RoboDK station: My_Bachelor_Project_Sim.rdk

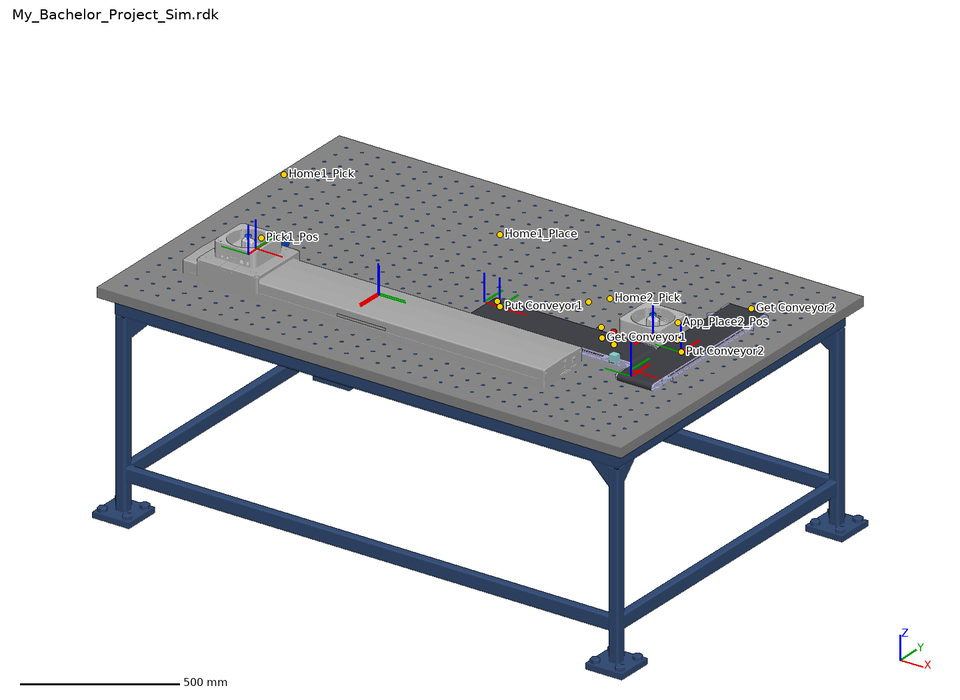
[picture v0: the station drawn from its stored meshes, robots at their saved joint values, targets as dots, program paths as lines]
Station My_Bachelor_Project_Sim (saved by RoboDK 5.9.2). Poses are relative to the parent item; angles as X-Y-Z fixed-axis rotations.
  - object Table  at (0, 0, 0) mm, size 2020 x 1340 x 800 mm, geometry from Table-2000x1200x800mm.sld
    - frame Conveyor1_frame at (730, -120, 40) mm
      - object Conveyor1 at (520, -80, -20) mm, rotated rx 0 ry 0 rz 90 deg, size 179.1 x 627.2 x 32.2 mm
      - frame Conveyor_1 Base at (0, 0, 0) mm
        - robot Conveyor_1: 1 axes
            modified DH rows (alpha deg, a mm, theta deg, d mm): 0, 0, 0, 0 linear
            base shift (0, 0, 0) mm, rotated rx 0 ry 90 rz 0 deg
            joint limits [0] to [600]; home [0]; saved at [0]
      - target Put Conveyor1 (Cartesian target) at (59.25, 0, -0.79) mm; joints [134.006, 22.86, -66.558, 43.699, -45.994, 0]
      - target Get Conveyor1 (Cartesian target) at (450, 0, 0) mm; joints [0, 0, 0, 0, 0, 43.699]
      - object Motion_Sensor at (450, 62, 20) mm, size 18 x 18 x 24 mm
      - object Colour_Sensor at (550, -108, -10) mm, size 25.9 x 25.9 x 25.9 mm, geometry from Cube-50mm (1).sld
      - frame Put_Conveyor1_Frame at (60, 0, 0) mm
        - target Home1_Place (Cartesian target) at (0, 0, 250) mm, rotated rx 180 ry 0 rz -90 deg; joints [0, 0, 0, 0] of Dobot Magician1
        - target Place1_Pos (Cartesian target) at (4.5, -22, 29.12) mm, rotated rx 180 ry 0 rz -90 deg; joints [-2.421, 65.885, 80.616, -2.421] of Dobot Magician1
    - frame Conveyor2_Frame at (1360, -220, 20) mm
      - frame Put_Conveyor2_Frame at (80, 160, 20) mm, rotated rx 0 ry 0 rz 90 deg
        - target Put Conveyor2 (Cartesian target) at (0, 0, 0) mm; joints [134.006, 22.86, -66.558, 43.699, -45.994, 0]
        - target Get Conveyor2 (Cartesian target) at (380, 0, 0) mm; joints [0, 0, 0, 0, 0, 43.699]
      - object Conveyor2 at (0, 0, 0) mm, size 179.1 x 627.2 x 32.2 mm
      - frame Conveyor_2 Base at (50, -70, 20) mm, rotated rx 0 ry 0 rz 90 deg
        - robot Conveyor_2: 1 axes
            modified DH rows (alpha deg, a mm, theta deg, d mm): 0, 0, 0, 0 linear
            base shift (0, 0, 0) mm, rotated rx 0 ry 90 rz 0 deg
            joint limits [0] to [600]; home [0]; saved at [380]
  - frame Rail_Reference at (480, -340, 90) mm, rotated rx 0 ry 0 rz -90 deg
    - frame Linear Rail Base at (10, 10, 0) mm
      - robot Linear Rail  (model Brooks PreciseFlex Linear Rail 1000): 1 axes
          modified DH rows (alpha deg, a mm, theta deg, d mm): 0, 0, 0, 0 linear
          base shift (0, 0, 0) mm, rotated rx 0 ry 90 rz 90 deg
          joint limits [-500] to [500]; home [0]; saved at [-500]
        - frame Dobot Magician1 Base at (0, 0, 1) mm, rotated rx 0 ry 0 rz -180 deg
          - robot Dobot Magician1 (model Dobot Magician): 4 axes, payload 0.5 kg, reach 320 mm, repeatability 0.2 mm, weight 4 kg
              joint limits [-90, -0.001, -10, -90] to [90, 85, 95, 90]; home [0, 0, 0, 0]; saved at [-26.105, 17.869, 35.082, 63.895]
            - tool Vacuum Gripper1, TCP at (0, 0, 65) mm, size 37.5 x 41.5 x 68.1 mm
      - target Rail_Home (Cartesian target) at (0, 0, 0) mm; joints [0] of Linear Rail 
      - target Rail_Pick_Pos (Cartesian target) at (0, -500, 0) mm; joints [-500] of Linear Rail 
      - target Rail_Place_Pos (Cartesian target) at (0, 295.7, 0) mm; joints [295.7] of Linear Rail 
  - frame Box_Frame at (-120, -150, 0) mm
    - object Red_Cube at (50, 0, 0) mm, size 25 x 25 x 25 mm, geometry from Cube-50mm (1).sld
    - object Green_Cube at (0, 50, 0) mm, size 25 x 25 x 25 mm, geometry from Cube-50mm (1).sld
    - object Blue_Cube at (50, 50, 0) mm, size 25 x 25 x 25 mm, geometry from Cube-50mm (1).sld
    - target Home1_Pick (Cartesian target) at (100, 10, 280) mm, rotated rx 180 ry 0 rz -90 deg; joints [2.726, 1.232, 5.453, 2.726] of Dobot Magician1
    - target Pick1_Pos (Cartesian target) at (13.34, 10.05, 37.21) mm, rotated rx 180 ry 0 rz -90 deg; joints [24.71, 81.254, 75.504, 24.71] of Dobot Magician1
    - object yellow_Cube at (0, 0, 0) mm, size 25 x 25 x 25 mm, geometry from Cube-50mm (1).sld
  - frame Dobot Magician2 Base at (1240, 70, 0) mm, rotated rx 0 ry 0 rz -90 deg
    - robot Dobot Magician2 (model Dobot Magician): 4 axes, payload 0.5 kg, reach 320 mm, repeatability 0.2 mm, weight 4 kg
        joint limits [-90, -0.001, -10, -90] to [90, 85, 95, 90]; home [0, 0, 0, 0]; saved at [0, 10.83, -4.63, 0]
      - tool Vacuum Gripper2, TCP at (0, 0, 65) mm, size 37.5 x 41.5 x 68.1 mm
    - target Home2_Pick (Cartesian target) at (232.89, 0, 212.46) mm, rotated rx 180 ry 0 rz -180 deg; joints [0, 10.83, -4.63, 0] of Dobot Magician2
    - target App_Pick2_Pos (Cartesian target) at (245.79, -71.87, 184.7) mm, rotated rx 180 ry 0 rz 163.7 deg; joints [-16.3, 21, 3.64, 0] of Dobot Magician2
    - target Pick2_Pos (Cartesian target) at (196.48, -57.46, 81.24) mm, rotated rx 180 ry 0 rz 163.7 deg; joints [-16.3, 21.33, 49.94, 0] of Dobot Magician2
    - target Sensor_Place2_Pos (Cartesian target) at (287.45, 53.95, 89.18) mm, rotated rx 180 ry 0 rz -169.37 deg; joints [10.63, 48.57, 27.62, 0] of Dobot Magician2
    - target App_Place2_Pos (Cartesian target) at (124.89, 185.02, 137.37) mm, rotated rx 180 ry 0 rz -124.02 deg; joints [55.98, 12.47, 25.14, 0] of Dobot Magician2
    - target Place2_Pos (Cartesian target) at (124.99, 180.37, 74.44) mm, rotated rx 180 ry 0 rz -124.72 deg; joints [55.28, 28.22, 49.94, 0] of Dobot Magician2
  - Python program Dobot_1_Prog (listed below)
  - Python program Dobot_2_Prog (listed below)
  - Python program Conveyor_1_Prog (listed below)
  - Python program Conveyor_2_Prog (listed below)
  - Python program Main_Common_Prog (listed below)

--- Python program Dobot_1_Prog ---
# Link to RoboDK
#### Dobot1 Programme ####

from robolink import *
from robodk import *
from time import sleep
sim = robolink.Robolink()

#Items
base = sim.Item("Dobot Magician1 Base")
robot1 = sim.Item("Dobot Magician1")
tool1 = sim.Item("Vacuum Gripper1")


#Conveyors
conveyor1 = sim.Item("Conveyor Belt1")


if not robot1.Valid():
    raise Exception("Robot not found")
if not tool1.Valid():
    raise Exception("Tool not found")

#frames
baseFrame = sim.Item("Dobot Magician1 Base")
rail = sim.Item("Linear Rail", ITEM_TYPE_ROBOT)
pickFrame =sim.Item("Box_Frame")
putFrame  = sim.Item("Put_Conveyor1_Frame")

# Targets
home1_Pick = sim.Item("Home1_Pick")
home1_Place = sim.Item("Home1_Place")
#app_Pick_Pos = sim.Item("App_Pick_Pos")
#app_Place_Pos = sim.Item("App__Place_Pos")
pick_Pos = sim.Item("Pick_Pos")
place_Pos = sim.Item("Place_Pos")

#objects
box1 = sim.Item("Yellow_Cube")
box2= sim.Item("Red_Cube")
box3 = sim.Item("Green_Cube")
box4 = sim.Item("Blue_Cube")
conveyor_Frame = sim.Item("Conveyro_Box_Frame")

# Targets (RAIL)

rail_home  = sim.Item("Rail_Home")
rail_pick  = sim.Item("Rail_Pick_Pos")
rail_place = sim.Item("Rail_Place_Pos")

for item in [rail_home, rail_pick, rail_place, app_pos_Pick, app_Pos_Place, pick_Pos, place_Pos]:
    if not item.Valid():
        raise Exception(f"Missing item: {item.Name()}")

robot1.setSpeed(200,50)
robot1.setPoseTool(tool1)

robot1.setPoseFrame(baseFrame)
rail.MoveJ(rail_home)
rail.MoveJ(rail_pick)

#Pick
robot1.setPoseFrame(pickFrame)
box.setParentStatic(pickFrame)
robot1.MoveJ(app_pos_Pick)
robot1.MoveJ(pick_Pos)
tool1.AttachClosest()
robot1.MoveJ(app_pos_Pick)

#Move to Put
robot1.setPoseFrame(baseFrame)
rail.MoveJ(rail_place)

#Put
robot1.setPoseFrame(putFrame)
robot1.MoveJ(app_Pos_Place)
robot1.MoveJ(place_Pos)
tool1.DetachAll()
box.setParent(putFrame)
box.setParentStatic(conveyor1)
robot1.MoveJ(app_Pos_Place)

robot1.setPoseFrame(baseFrame)
rail.MoveJ(rail_home)

--- Python program Dobot_2_Prog ---
from robolink import *
from robodk import *
sim = robolink.Robolink()

#Items
base2 = sim.Item("Dobot Magician2 Base")
robot2 = sim.Item("Dobot Magician2")
tool2  = sim.Item("Vacuum Gripper2")
conveyor1 = sim.Item("Conveyor1")
conveyor2 = sim.Item("Conveyor")
box = sim.Item("Cube_Box")

# Frames
box_Frame_Pick = sim.Item("Conv1_Box_Frame")
box_Frame_Put = sim.Item("Conv2_Box_Frame")

# Targets
home2 = sim.Item("Home_Dobot2")
app_Pick_Conv1 = sim.Item("App_Pick_Pose_Conv1")
Pick_Conv1 = sim.Item("Pick_Pos_Conv1")
app_put_Conv2 = sim.Item("App_Put_Box_Conv2")
put_Conv2 = sim.Item("Put_Box_Conv2")


base = sim.Item("Dobot Magician2 Base")

# Gå to the conveyor and pick the cube

robot2.setSpeed(200,50)

# go to home for dobot2 base frame
robot2.setFrame(base2)
robot2.MoveJ(home2)

# go to pick position
robot2.setTool(tool2)
robot2.setFrame(base2)
robot2.MoveJ(app_Pick_Conv1)
robot2.MoveJ(Pick_Conv1)

# attach cube
box.setParent(box_Frame_Pick)
tool2.AttachClosest()

# go to put position
robot2.MoveJ(app_put_Conv2)
robot2.MoveJ(put_Conv2)
box.setParent(conveyor2)
tool2.DetachAll()

robot2.setFrame(base2)
robot2.MoveJ(home2)

--- Python program Conveyor_1_Prog ---
#### Conveyor1 programme ####

# To connect with the RoboDK
from robolink import *
from robodk import *
from time import sleep

sim = robolink.Robolink()

# Item
conveyor1 = sim.Item("Conveyor Belt1")
box = sim.Item("Cube")

# Frame
conveyor1_Frame = sim.Item("Conveyor Belt1 Base")
conveyorReference = sim.Item("ConveyorReference")
put_Conveyor1_Frame = sim.Item("Put_Conveyor1_Frame", ITEM_TYPE_FRAME)

# Targets
put_pos = sim.Item("Put Conveyor1")
get_pos = sim.Item("Get Conveyor1")

if not conveyor1.Valid() or not box.Valid():
    raise Exception("Items not found")

# Programme to set or atach the box ti the put_pos
# Attach cube to Put Conveyor1

all_items = sim.ItemList()
for item in all_items:
    print(item.Name())

def run_cycle():

    if not put_Conveyor1_Frame.Valid():
        raise Exception("Put_Conveyor1_Frame not found")

    box.setParentStatic(put_Conveyor1_Frame)
    box.setPose(transl(0,0,0,))

    box.setParentStatic(conveyor1)
    sleep(0.1)

     # Move conveyor slowly
    for i in range(0,1500,20):   # step size controls speed
        conveyor1.setJoints([i])
        sleep(0.05)
    print("Conveyor1 cycle complete")

 # Run 5 times again
print("Starting 5-run loop...")
for i in range(2):
    print(f"Iteration {i+1}")
    run_cycle()
    sleep(0.5)

--- Python program Conveyor_2_Prog ---
#### Conveyor2 programme ####

# To connect with the RoboDK
from robolink import *
from robodk import *
from time import sleep

sim = robolink.Robolink()

# Item
conveyor2 = sim.Item("Conveyor Belt2")
box_frame = sim.Item("Put_Conv2")
box = sim.Item("Cube_Box")

# Check validity
if not box.Valid():
    raise Exception("Check! cube not found")

#Targets
home_pos = sim.Item("Conv2_Home_Put")
yellow_pos = sim.Item("Get_Conv2_Yellow")
non_yellow_pos =sim.Item("Get_Conv2_Non_Yellow")

if not home_pos.Valid() or not yellow_pos.Valid() or not non_yellow_pos.Valid():
    raise Exception("Check target names")

# Reset conveyor
box.setParentStatic(conveyor2)
sleep(0.1)

#conveyor2.MoveJ(home_pos)
#sleep(0.3)
cube_colour = "yellow"
#cube_colour = "red"
#cube_colour = "green"
#cube_colour = "blue"


# Move depending on colour
if cube_colour == "yellow":
    conveyor2.MoveJ(yellow_pos)
else:
    conveyor2.MoveJ(non_yellow_pos)

sleep(0.5)

conveyor2.MoveJ(home_pos)

--- Python program Main_Common_Prog ---
### Main programme

# To connect with the RoboDK
from robolink import *
from robodk import *
from time import sleep

sim = robolink.Robolink()
